# EPICS IOC start-up script: iocsh/ethercatmcAuxBitsStatus.iocsh
dbLoadRecords("ethercatmcAuxBitsStatus.template", "P=$(P), R=$(R), AXIS_NO=$(AXIS_NO), MOTOR_PORT=$(MOTOR_PORT), ASYN_PORT=$(ASYN_PORT), AXIS_NO=$(AXIS_NO), DESC=$(DESC), PREC=$(PREC) ")
